FUNCTION_BLOCK FB_TP (* standard timer function block (pulse) *)
  (* Standard: 61131-3; Classification: standard timer function block *)
  (* Version 1.0, 2009-09-14, 4DIAC-IDE, 4DIAC-Consortium *)
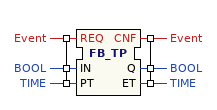
  EVENT_INPUT
    REQ WITH IN, PT; (* Service Request *)
  END_EVENT
  EVENT_OUTPUT
    CNF WITH Q, ET; (* Confirmation of Requested Service *)
  END_EVENT
  VAR_INPUT
    IN : BOOL; (* Input *)
    PT : TIME; (* Pulse time *)
  END_VAR
  VAR_OUTPUT
    Q : BOOL; (* output *)
    ET : TIME; (* elapse time *)
  END_VAR
  (* Service APPLICATION/RESOURCE: standard timer function block (pulse) *)
END_FUNCTION_BLOCK
